// TIA Portal V17 export
// export: Created 2023-12-22T15:08:09.7281351Z, ExportSetting WithDefaults, DisplayName Totally Integrated Automation Portal, DisplayVersion V17, DisplayName TIA Portal Openness, DisplayVersion V17, DisplayName TIA Portal Version Control Interface, DisplayVersion V17, DisplayName STEP 7 Professional, DisplayVersion V17, DisplayName STEP 7 Safety, DisplayVersion V17, DisplayName WinCC Advanced, DisplayVersion V17
DATA_BLOCK "Supp_DB"   // DB4
VERSION : 0.1
// stored: AutoNumber true, DBAccessibleFromOPCUA true, DBAccessibleFromWebserver true, InstanceOfName Support, InstanceOfType FB
"Support"
   // VAR
   //    pipe_in : Array[0..20] of Int;
   //    pipe_out : Array[0..20] of Int;
   //    state : Array[0..15] of Bool;
   // END_VAR
BEGIN
END_DATA_BLOCK
